// TwinCAT 3 PLC project code
// ProgramVersion: 3.1.4024.0
// libraries:
//   Tc2_Standard, * (Beckhoff Automation GmbH)
//   Tc2_System, * (Beckhoff Automation GmbH)
//   Tc3_Module, * (Beckhoff Automation GmbH)
// project tree:
//   DUTs/ dt_Parameters.TcDUT
//   GVLs/ Parameters.TcGVL
//   / PlcTask.TcTTO
//   POUs/ FB_Outer.TcPOU, FB_Middler.TcPOU, FB_Inner.TcPOU, FB_Parameters_Base.TcPOU, FB_Parameters_Store.TcPOU, If_Parameters.TcIO, MAIN.TcPOU
// real-time tasks:
//   TASK PlcTask: cycle T#10ms, priority 20, ADS port 350
//   TASK PlcTask1: cycle T#10ms, priority 21, ADS port 351

CONFIGURATION code
    RESOURCE PLC ON TwinCAT3
        TASK PlcTask(INTERVAL := T#10ms, PRIORITY := 21);
        PROGRAM MAIN WITH PlcTask : MAIN;
    END_RESOURCE
END_CONFIGURATION

// ---- DUTs/dt_Parameters.TcDUT
TYPE dt_Parameters :
STRUCT
	Scale	: LREAL;
	Etc		: INT;
END_STRUCT
END_TYPE

// ---- GVLs/Parameters.TcGVL
{attribute 'qualified_only'}
VAR_GLOBAL
	Parameters	: FB_Parameters_Store	:= (Pars := (
											Scale := 3.14,
											Etc := 42
										));
END_VAR

// ---- POUs/If_Parameters.TcIO
INTERFACE If_Parameters

PROPERTY Par : REFERENCE TO dt_Parameters
GET
END_GET
END_PROPERTY

END_INTERFACE

// ---- POUs/MAIN.TcPOU
PROGRAM MAIN
VAR
	outer	: FB_Outer(Parameters.Parameters);
END_VAR

END_PROGRAM

// ---- POUs/FB_Outer.TcPOU
FUNCTION_BLOCK FB_Outer EXTENDS FB_Parameters_Base
VAR
	middler	: FB_Middler(THIS^);
END_VAR

END_FUNCTION_BLOCK

// ---- POUs/FB_Parameters_Base.TcPOU
FUNCTION_BLOCK ABSTRACT FB_Parameters_Base IMPLEMENTS If_Parameters
VAR
	_par_ref_for_inner_use	: REFERENCE TO dt_parameters;
	_init_index				: UINT; //intialization order track
END_VAR
VAR_STAT
	_next_init_index		: UINT;
END_VAR

METHOD FB_init : BOOL
VAR_INPUT
	bInitRetains : BOOL; // if TRUE, the retain variables are initialized (warm start / cold start)
	bInCopyCode : BOOL;  // if TRUE, the instance afterwards gets moved into the copy code (online change)
	iParameters : If_Parameters;
END_VAR

_par_ref_for_inner_use REF= iParameters.Par;

_init_index := _next_init_index;
_next_init_index := _next_init_index + 1;
END_METHOD

PROPERTY Par : REFERENCE TO dt_Parameters
GET

Par REF= _par_ref_for_inner_use;
END_GET
END_PROPERTY

END_FUNCTION_BLOCK

// ---- POUs/FB_Middler.TcPOU
FUNCTION_BLOCK FB_Middler EXTENDS FB_Parameters_Base
VAR
	inner	: FB_Inner(THIS^);
END_VAR

END_FUNCTION_BLOCK

// ---- POUs/FB_Inner.TcPOU
FUNCTION_BLOCK FB_Inner EXTENDS FB_Parameters_Base
VAR_INPUT
END_VAR
VAR_OUTPUT
END_VAR
VAR
END_VAR

END_FUNCTION_BLOCK

// ---- POUs/FB_Parameters_Store.TcPOU
FUNCTION_BLOCK FB_Parameters_Store IMPLEMENTS If_Parameters
VAR_INPUT PERSISTENT
	Pars	: dt_Parameters;
END_VAR

PROPERTY Par : REFERENCE TO dt_Parameters
GET

Par REF= Pars;
END_GET
END_PROPERTY

END_FUNCTION_BLOCK
